FUNCTION_BLOCK SAMPLE_UINT (* Sample a single UINT - see SAMPLE_1 *)
  (* Standard: 61499-1; Classification: Math; Function: Sampling; Type: UINT *)
  (* Version 0.0, 2006-05-28, JHC, Holobloc Inc *)
  (* Compiler header: package fb.rt.math; *)
  (* Compiler Java Sun JDK 1.5.0 *)
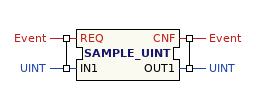
  EVENT_INPUT
    REQ WITH IN1; (* Request to Sample with Monitor Lock *)
  END_EVENT
  EVENT_OUTPUT
    CNF WITH OUT1; (* Initial Sample or OUT1 changed *)
  END_EVENT
  VAR_INPUT
    IN1 : UINT; (* Data to Sample *)
  END_VAR
  VAR_OUTPUT
    OUT1 : UINT; (* Sampled Data *)
  END_VAR
END_FUNCTION_BLOCK
